(* IEC 61131-3 sources: JaccoSigma/tempclass/Class/My_ReadClass, 1 file *)

(* ---- My_ReadClass.st ---- *)
(*!
<Class
	Name               = "My_ReadClass"
	Revision           = "0.0"
	RealtimeTask       = "false"
	CyclicTask         = "true"
	DefCyclictime      = "1 ms"
	BackgroundTask     = "false"
	Sigmatek           = "false"
	OSInterface        = "false"
	HighPriority       = "false"
	Automatic          = "false"
	UpdateMode         = "Prescan"
	SharedCommandTable = "true"
	Objectsize         = "(490,120)">
	<Channels>
		<Server Name="ReadCyclic" Visualized="false" Initialize="false" WriteProtected="false" Retentive="false"/>
		<Server Name="ReadWriteOnce" Visualized="false" Initialize="false" WriteProtected="false" Retentive="false"/>
		<Server Name="WriteServer" Visualized="false" Initialize="false" WriteProtected="false" Retentive="false"/>
		<Client Name="ReadClient" Required="false" Internal="false"/>
	</Channels>
</Class>
*)
My_ReadClass : CLASS
  //Servers:
	ReadWriteOnce 	: SvrChCmd_DINT;
	ReadCyclic 	: SvrCh_DINT;
	WriteServer 	: SvrCh_DINT;
  //Clients:
	ReadClient 	: CltCh_DINT;
  //Variables:
  //Functions:

	FUNCTION VIRTUAL GLOBAL CyWork
		VAR_INPUT
			EAX 	: UDINT;
		END_VAR
		VAR_OUTPUT
			state (EAX) 	: UDINT;
		END_VAR;

	FUNCTION VIRTUAL GLOBAL ReadWriteOnce::Write
		VAR_INPUT
			input (EAX) 	: DINT;
		END_VAR
		VAR_OUTPUT
			result (EAX) 	: DINT;
		END_VAR;

	FUNCTION VIRTUAL GLOBAL WriteServer::Write
		VAR_INPUT
			input (EAX) 	: DINT;
		END_VAR
		VAR_OUTPUT
			result (EAX) 	: DINT;
		END_VAR;
  //Tables:
	FUNCTION @STD
		VAR_OUTPUT
			ret_code	: CONFSTATES;
		END_VAR;
	FUNCTION GLOBAL TAB @CT_;
END_CLASS;

FUNCTION VIRTUAL GLOBAL My_ReadClass::ReadWriteOnce::Write
	VAR_INPUT
		input (EAX) 	: DINT;
	END_VAR
	VAR_OUTPUT
		result (EAX) 	: DINT;
	END_VAR

	ReadWriteOnce := input;

//  ReadClient := ReadClient.Read();
  WriteServer.Write(input:=WriteServer);

	result := ReadWriteOnce := 0;

END_FUNCTION

FUNCTION VIRTUAL GLOBAL My_ReadClass::CyWork
	VAR_INPUT
		EAX 	: UDINT;
	END_VAR
	VAR_OUTPUT
		state (EAX) 	: UDINT;
	END_VAR

  if ReadCyclic = 1 then
    ReadClient := ReadClient.Read();
  end_if;

  if ReadCyclic = 2 then
    WriteServer.Write(input:=WriteServer);
  end_if;

	state := READY;

END_FUNCTION

FUNCTION VIRTUAL GLOBAL My_ReadClass::WriteServer::Write
	VAR_INPUT
		input (EAX) 	: DINT;
	END_VAR
	VAR_OUTPUT
		result (EAX) 	: DINT;
	END_VAR

	WriteServer := input;

	result := WriteServer;

END_FUNCTION
